PROGRAM Stn5
VAR

	start5: BOOL;
	reset5: BOOL;

	Stn5ProcessFE: F_TRIG;
	Stn5ProcessRE: R_TRIG;
	bCutStn5ProcessHalt: BOOL;
	DoorClose5: R_TRIG;
	bStn5DoorClamp: BOOL;

END_VAR
VAR // added by the converter: edge detectors and wires of the graphical bodies
    _w1, _w2 : ANY;
END_VAR

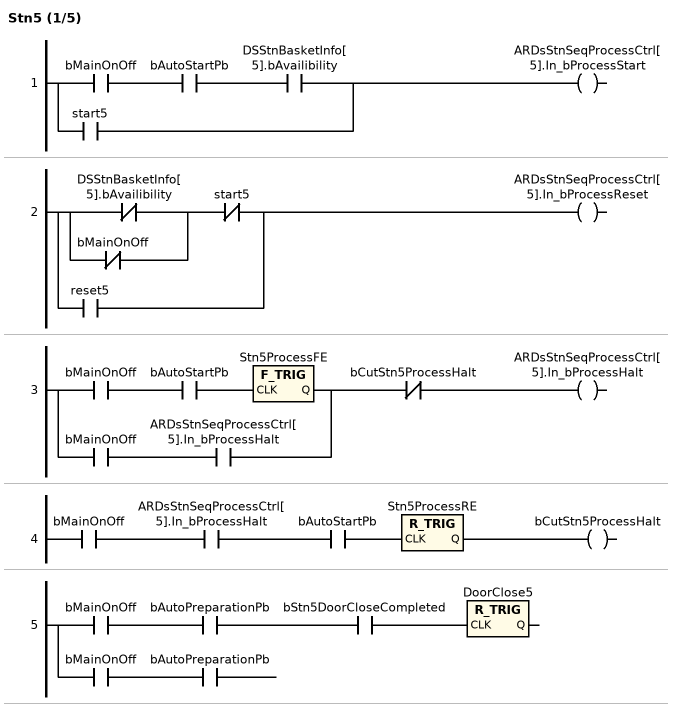
// NETWORK 1
ARDsStnSeqProcessCtrl[5].In_bProcessStart := bMainOnOff AND bAutoStartPb AND DSStnBasketInfo[5].bAvailibility OR start5;

// NETWORK 2
ARDsStnSeqProcessCtrl[5].In_bProcessReset := (NOT DSStnBasketInfo[5].bAvailibility OR NOT bMainOnOff) AND NOT start5 OR reset5;

// NETWORK 3
Stn5ProcessFE(CLK := bMainOnOff AND bAutoStartPb); // F_TRIG
ARDsStnSeqProcessCtrl[5].In_bProcessHalt := (Stn5ProcessFE.Q OR bMainOnOff AND ARDsStnSeqProcessCtrl[5].In_bProcessHalt) AND NOT bCutStn5ProcessHalt;

// NETWORK 4
Stn5ProcessRE(CLK := bMainOnOff AND ARDsStnSeqProcessCtrl[5].In_bProcessHalt AND bAutoStartPb); // R_TRIG
bCutStn5ProcessHalt := Stn5ProcessRE.Q;

// NETWORK 5
DoorClose5(CLK := bMainOnOff AND bAutoPreparationPb AND bStn5DoorCloseCompleted); // R_TRIG
(* DoorClose5.Q OR bMainOnOff AND bAutoPreparationPb; result not used *)

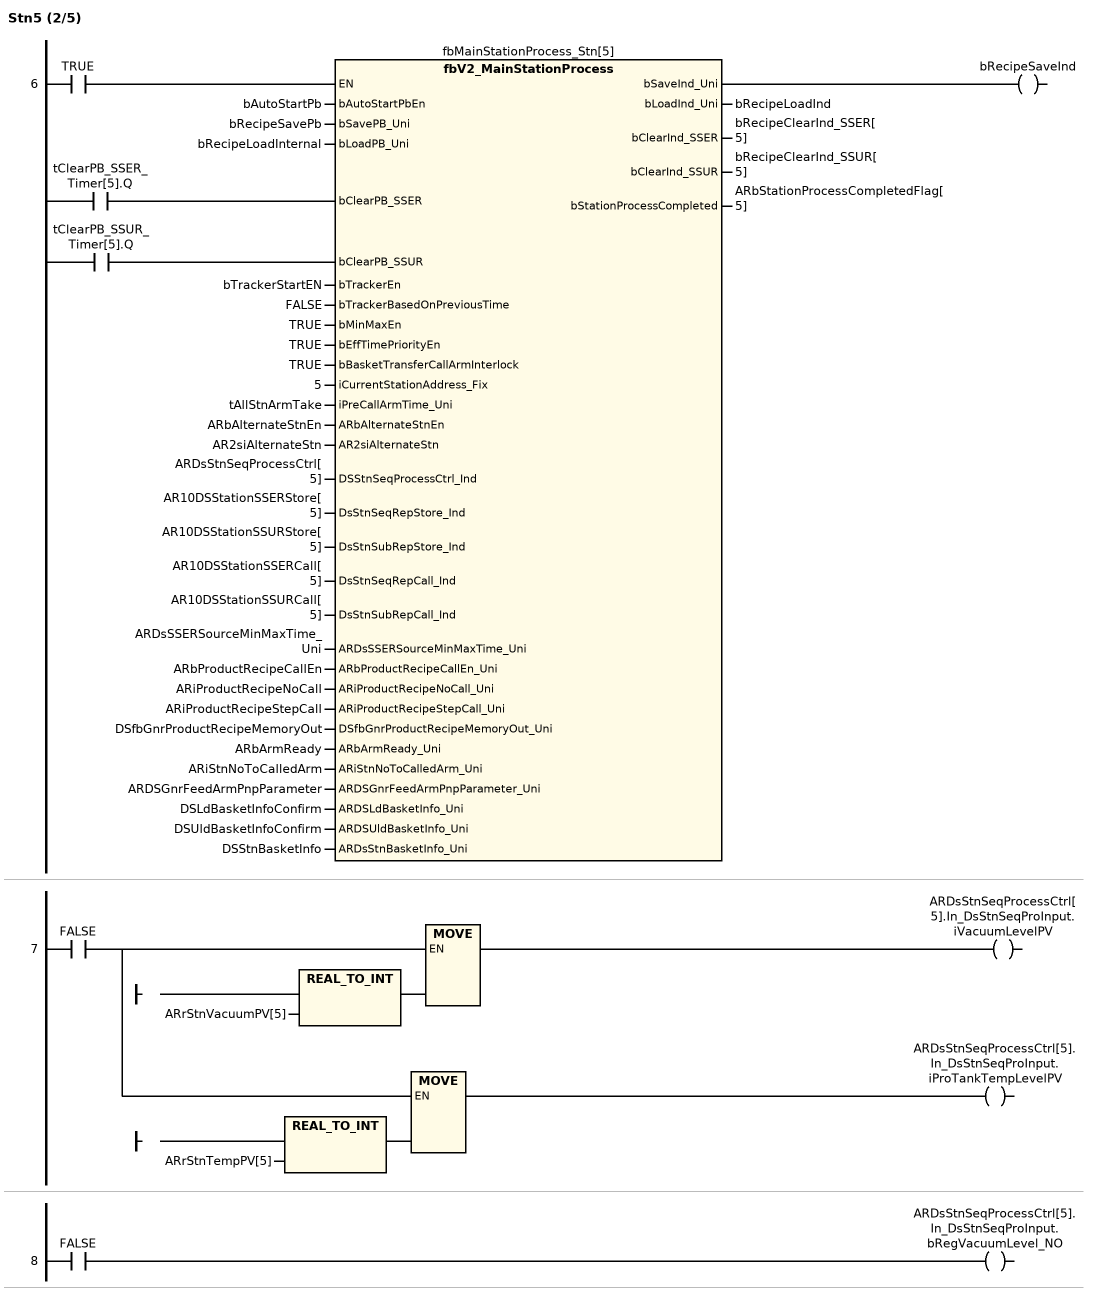
// NETWORK 6
fbMainStationProcess_Stn[5](
    bAutoStartPbEn := bAutoStartPb,
    bSavePB_Uni := bRecipeSavePb,
    bLoadPB_Uni := bRecipeLoadInternal,
    bClearPB_SSER := tClearPB_SSER_Timer[5].Q,
    bClearPB_SSUR := tClearPB_SSUR_Timer[5].Q,
    bTrackerEn := bTrackerStartEN,
    bTrackerBasedOnPreviousTime := FALSE,
    bMinMaxEn := TRUE,
    bEffTimePriorityEn := TRUE,
    bBasketTransferCallArmInterlock := TRUE,
    iCurrentStationAddress_Fix := 5,
    iPreCallArmTime_Uni := tAllStnArmTake,
    ARbAlternateStnEn := ARbAlternateStnEn,
    AR2siAlternateStn := AR2siAlternateStn,
    DSStnSeqProcessCtrl_Ind := ARDsStnSeqProcessCtrl[5],
    DsStnSeqRepStore_Ind := AR10DSStationSSERStore[5],
    DsStnSubRepStore_Ind := AR10DSStationSSURStore[5],
    DsStnSeqRepCall_Ind := AR10DSStationSSERCall[5],
    DsStnSubRepCall_Ind := AR10DSStationSSURCall[5],
    ARDsSSERSourceMinMaxTime_Uni := ARDsSSERSourceMinMaxTime_Uni,
    ARbProductRecipeCallEn_Uni := ARbProductRecipeCallEn,
    ARiProductRecipeNoCall_Uni := ARiProductRecipeNoCall,
    ARiProductRecipeStepCall_Uni := ARiProductRecipeStepCall,
    DSfbGnrProductRecipeMemoryOut_Uni := DSfbGnrProductRecipeMemoryOut,
    ARbArmReady_Uni := ARbArmReady,
    ARiStnNoToCalledArm_Uni := ARiStnNoToCalledArm,
    ARDSGnrFeedArmPnpParameter_Uni := ARDSGnrFeedArmPnpParameter,
    ARDSLdBasketInfo_Uni := DSLdBasketInfoConfirm,
    ARDSUldBasketInfo_Uni := DSUldBasketInfoConfirm,
    ARDsStnBasketInfo_Uni := DSStnBasketInfo,
    bLoadInd_Uni => bRecipeLoadInd,
    bClearInd_SSER => bRecipeClearInd_SSER[5],
    bClearInd_SSUR => bRecipeClearInd_SSUR[5],
    bStationProcessCompleted => ARbStationProcessCompletedFlag[5]); // fbV2_MainStationProcess
bRecipeSaveInd := fbMainStationProcess_Stn[5].bSaveInd_Uni;

// NETWORK 7
IF FALSE THEN _w1 := REAL_TO_INT(ARrStnVacuumPV[5]); END_IF
ARDsStnSeqProcessCtrl[5].In_DsStnSeqProInput.iVacuumLevelPV := _w1;
IF FALSE THEN _w2 := REAL_TO_INT(ARrStnTempPV[5]); END_IF
ARDsStnSeqProcessCtrl[5].In_DsStnSeqProInput.iProTankTempLevelPV := _w2;

// NETWORK 8
ARDsStnSeqProcessCtrl[5].In_DsStnSeqProInput.bRegVacuumLevel_NO := FALSE;

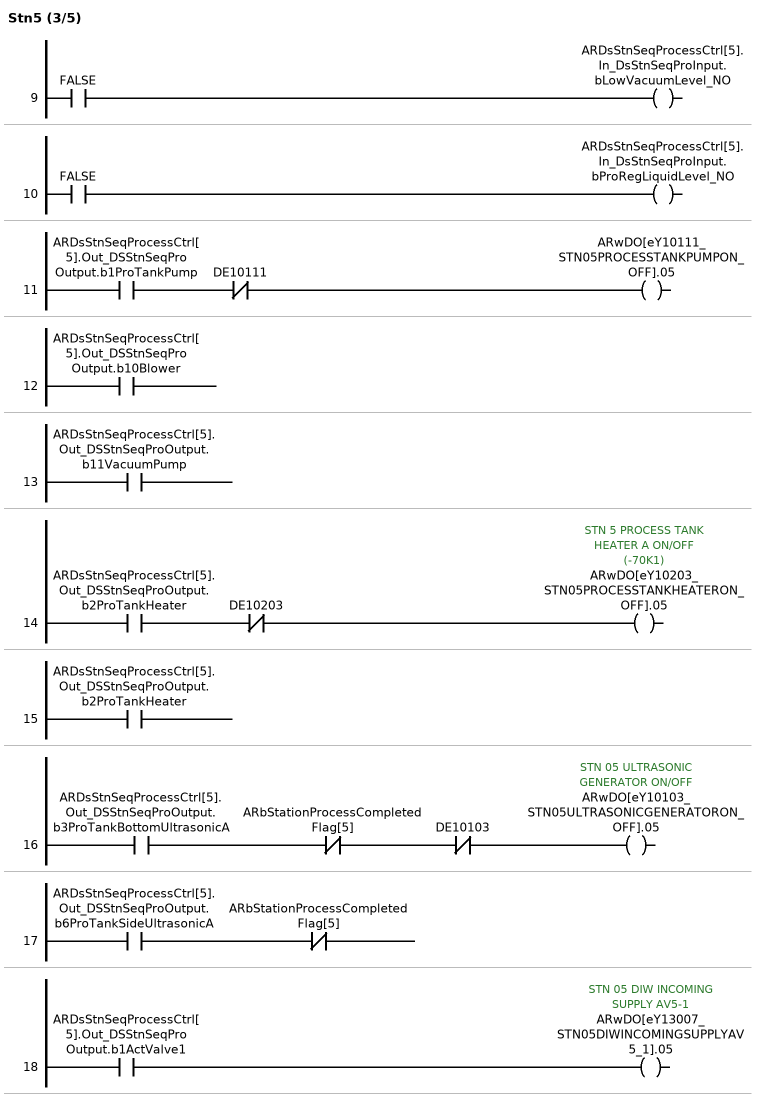
// NETWORK 9
ARDsStnSeqProcessCtrl[5].In_DsStnSeqProInput.bLowVacuumLevel_NO := FALSE;

// NETWORK 10
ARDsStnSeqProcessCtrl[5].In_DsStnSeqProInput.bProRegLiquidLevel_NO := FALSE;

// NETWORK 11
ARwDO[eY10111_STN05PROCESSTANKPUMPON_OFF].05 := ARDsStnSeqProcessCtrl[5].Out_DSStnSeqProOutput.b1ProTankPump AND NOT DE10111;

// NETWORK 12
(* ARDsStnSeqProcessCtrl[5].Out_DSStnSeqProOutput.b10Blower; not connected *)

// NETWORK 13
(* ARDsStnSeqProcessCtrl[5].Out_DSStnSeqProOutput.b11VacuumPump; not connected *)

// NETWORK 14
//   ARwDO[eY10203_STN05PROCESSTANKHEATERON_OFF].05: STN 5 PROCESS TANK HEATER A ON/OFF (-70K1)
ARwDO[eY10203_STN05PROCESSTANKHEATERON_OFF].05 := ARDsStnSeqProcessCtrl[5].Out_DSStnSeqProOutput.b2ProTankHeater AND NOT DE10203;

// NETWORK 15
(* ARDsStnSeqProcessCtrl[5].Out_DSStnSeqProOutput.b2ProTankHeater; not connected *)

// NETWORK 16
//   ARwDO[eY10103_STN05ULTRASONICGENERATORON_OFF].05: STN 05 ULTRASONIC GENERATOR ON/OFF
ARwDO[eY10103_STN05ULTRASONICGENERATORON_OFF].05 := ARDsStnSeqProcessCtrl[5].Out_DSStnSeqProOutput.b3ProTankBottomUltrasonicA AND NOT ARbStationProcessCompletedFlag[5] AND NOT DE10103;

// NETWORK 17
(* ARDsStnSeqProcessCtrl[5].Out_DSStnSeqProOutput.b6ProTankSideUltrasonicA AND NOT ARbStationProcessCompletedFlag[5]; result not used *)

// NETWORK 18
//   ARwDO[eY13007_STN05DIWINCOMINGSUPPLYAV5_1].05: STN 05 DIW INCOMING SUPPLY AV5-1
ARwDO[eY13007_STN05DIWINCOMINGSUPPLYAV5_1].05 := ARDsStnSeqProcessCtrl[5].Out_DSStnSeqProOutput.b1ActValve1;

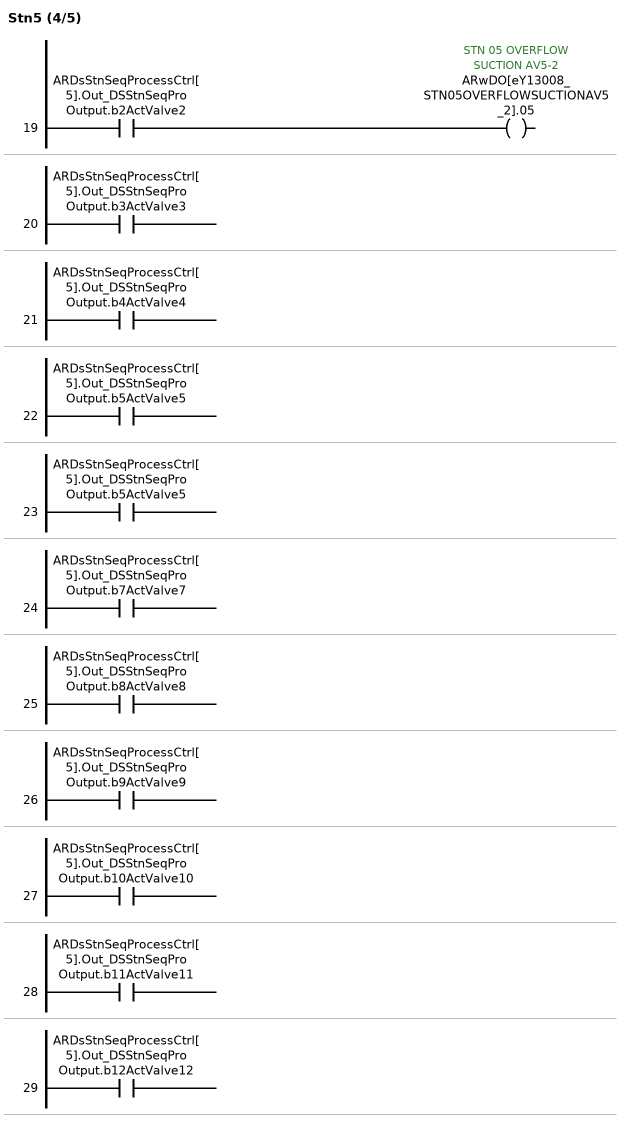
// NETWORK 19
//   ARwDO[eY13008_STN05OVERFLOWSUCTIONAV5_2].05: STN 05 OVERFLOW SUCTION AV5-2
ARwDO[eY13008_STN05OVERFLOWSUCTIONAV5_2].05 := ARDsStnSeqProcessCtrl[5].Out_DSStnSeqProOutput.b2ActValve2;

// NETWORK 20
(* ARDsStnSeqProcessCtrl[5].Out_DSStnSeqProOutput.b3ActValve3; not connected *)

// NETWORK 21
(* ARDsStnSeqProcessCtrl[5].Out_DSStnSeqProOutput.b4ActValve4; not connected *)

// NETWORK 22
(* ARDsStnSeqProcessCtrl[5].Out_DSStnSeqProOutput.b5ActValve5; not connected *)

// NETWORK 23
(* ARDsStnSeqProcessCtrl[5].Out_DSStnSeqProOutput.b5ActValve5; not connected *)

// NETWORK 24
(* ARDsStnSeqProcessCtrl[5].Out_DSStnSeqProOutput.b7ActValve7; not connected *)

// NETWORK 25
(* ARDsStnSeqProcessCtrl[5].Out_DSStnSeqProOutput.b8ActValve8; not connected *)

// NETWORK 26
(* ARDsStnSeqProcessCtrl[5].Out_DSStnSeqProOutput.b9ActValve9; not connected *)

// NETWORK 27
(* ARDsStnSeqProcessCtrl[5].Out_DSStnSeqProOutput.b10ActValve10; not connected *)

// NETWORK 28
(* ARDsStnSeqProcessCtrl[5].Out_DSStnSeqProOutput.b11ActValve11; not connected *)

// NETWORK 29
(* ARDsStnSeqProcessCtrl[5].Out_DSStnSeqProOutput.b12ActValve12; not connected *)

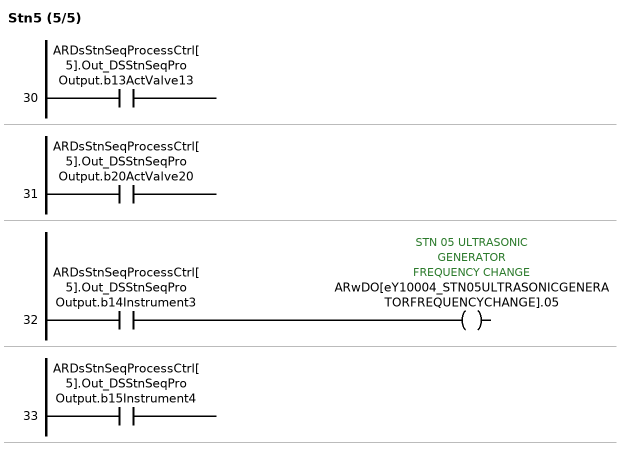
// NETWORK 30
(* ARDsStnSeqProcessCtrl[5].Out_DSStnSeqProOutput.b13ActValve13; not connected *)

// NETWORK 31
(* ARDsStnSeqProcessCtrl[5].Out_DSStnSeqProOutput.b20ActValve20; not connected *)

// NETWORK 32
//   ARwDO[eY10004_STN05ULTRASONICGENERATORFREQUENCYCHANGE].05: STN 05 ULTRASONIC GENERATOR FREQUENCY CHANGE
ARwDO[eY10004_STN05ULTRASONICGENERATORFREQUENCYCHANGE].05 := ARDsStnSeqProcessCtrl[5].Out_DSStnSeqProOutput.b14Instrument3;

// NETWORK 33
(* ARDsStnSeqProcessCtrl[5].Out_DSStnSeqProOutput.b15Instrument4; not connected *)

END_PROGRAM

(* stored: Version 1.1.0.1, ProductVersion 3.1.4024.12
   POU Stn5: Id {4b729fbe-d6fa-42fc-b2f4-c9dbafb52bfb}, SpecialFunc None *)
